# EPICS substitutions: iocs/MC03/MCApp/Db/SAI_save_restoreStatus.substitutions
file /opt/epics/modules/genericScan/db/save_restoreStatus.template {
pattern
{ DEVICE}
	{ "FMBGSCAN" }
}
# DEVICE: device name
